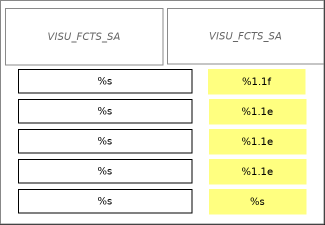
VISUALIZATION SA_REGUL_GAZ  // 325x225
VAR_IN_OUT
	m_Input_REGULATION : BLOCK_REGUL_PR_GAZ;
	m_Input_MACHINE : BLOCK_MODE_MARCHE_V2_0;
END_VAR
    Rectangle (0,0 325x225)
    Frame (5,8 158x57)
        shows VISU_FCTS_SA(m_Input_ID_XML := 29, m_Input_Operation := m_Input_REGULATION.OP_MARCHE, m_Input_UserRight := Global_Variables.PRG_USER.ACTU_USER.FONCTION_SA AND NOT m_Input_MACHINE.STATE_PROD)
    RoundedRectangle (18,69 174x24), "%s", text list: 'TextList_Gaz', text index: 15
    RoundedRectangle (208,69 97x25), "%1.1f", text variable: m_Input_REGULATION.PRM_Pos_Vanne, input disabled if: ((NOT PRG_User.ACTU_USER.FONCTION_SA AND NOT m_Input_MACHINE.STATE_PROD) OR (NOT PRG_User.ACTU_USER.MODIF_ENLIGNE AND m_Input_MACHINE.STATE_PROD)) <> 0
        OnMouseDown: write the text variable via InputWithLimits, min 0, max 100
    Frame (167,8 157x56)
        shows VISU_FCTS_SA(m_Input_ID_XML := 7, m_Input_Operation := m_Input_REGULATION.OP_ARRET, m_Input_UserRight := Global_Variables.PRG_USER.ACTU_USER.FONCTION_SA AND NOT m_Input_MACHINE.STATE_PROD)
    RoundedRectangle (18,99 174x24), "%s", text list: 'TextList_Gaz', text index: 16
    RoundedRectangle (209,99 97x25), "%1.1e", text variable: m_Input_REGULATION.PRM_Pressure, input disabled if: ((NOT PRG_User.ACTU_USER.FONCTION_SA AND NOT m_Input_MACHINE.STATE_PROD) OR (NOT PRG_User.ACTU_USER.MODIF_ENLIGNE AND m_Input_MACHINE.STATE_PROD)) <> 0
        OnMouseDown: write the text variable via InputWithLimits, min 0, max 1000
    RoundedRectangle (18,129 174x24), "%s", text list: 'TextList_Gaz', text index: 17
    RoundedRectangle (209,129 97x25), "%1.1e", text variable: m_Input_REGULATION.PRM_Pressure_L, input disabled if: ((NOT PRG_User.ACTU_USER.FONCTION_SA AND NOT m_Input_MACHINE.STATE_PROD) OR (NOT PRG_User.ACTU_USER.MODIF_ENLIGNE AND m_Input_MACHINE.STATE_PROD)) <> 0
        OnMouseDown: write the text variable via InputWithLimits, min 0, max 1000
    RoundedRectangle (18,159 174x24), "%s", text list: 'TextList_Gaz', text index: 18
    RoundedRectangle (209,159 97x25), "%1.1e", text variable: m_Input_REGULATION.PRM_Pressure_H, input disabled if: ((NOT PRG_User.ACTU_USER.FONCTION_SA AND NOT m_Input_MACHINE.STATE_PROD) OR (NOT PRG_User.ACTU_USER.MODIF_ENLIGNE AND m_Input_MACHINE.STATE_PROD)) <> 0
        OnMouseDown: write the text variable via InputWithLimits, min 0, max 1000
    RoundedRectangle (18,189 174x24), "%s", text list: 'TextList_Gaz', text index: 19
    RoundedRectangle (209,189 97x25), "%s", text variable: m_Input_REGULATION.PRM_Tim_Stab, input disabled if: ((NOT PRG_User.ACTU_USER.FONCTION_SA AND NOT m_Input_MACHINE.STATE_PROD) OR (NOT PRG_User.ACTU_USER.MODIF_ENLIGNE AND m_Input_MACHINE.STATE_PROD)) <> 0
        OnMouseDown: write the text variable via InputWithLimits
END_VISUALIZATION

(* stored: Version 1.1.0.1, ProductVersion 3.1.4024.10
   Visu SA_REGUL_GAZ: Id {efe4d5fd-ff96-4aa9-971a-01a92340a429} *)
